PROGRAM SavePersistent
///////////////////
// Save persistent data regularly
///////////////////
VAR
	FB_WritePersistentData : WritePersistentData  ;
	
	LTP2: TP;
	ClockPersistent: BOOL;
END_VAR

// WRITING CLOCK //
	LTP2(IN:=NOT LTP2.Q , PT:= T#1M);
	ClockPersistent := LTP2.Q;

FB_WritePersistentData(
						NETID:='', 
						PORT:= 851 ,
						START :=  ClockPersistent AND NOT FB_WritePersistentData.BUSY , 
						TMOUT := T#10S ) ;

END_PROGRAM

(* stored: Version 1.1.0.1, ProductVersion 3.1.4024.6
   POU SavePersistent: Id {1952dfde-46c3-44d7-a6d7-00d979227d56}, SpecialFunc None *)
